ABB RobotStudio station: Material Handeling (First Class) (5-3-2024)@7020.rsstn

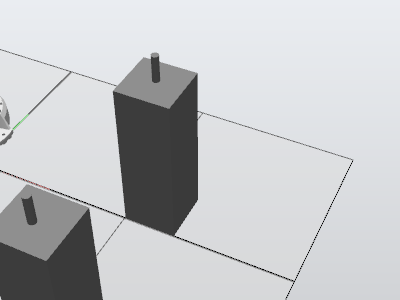
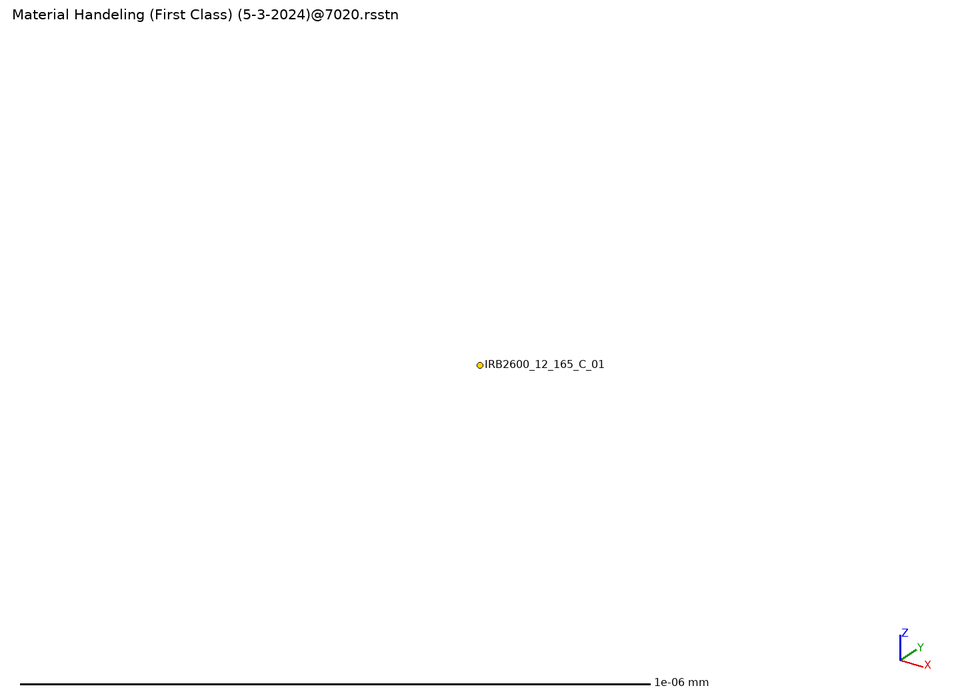
[picture v1: parts stored in the station drawn from their meshes, with robot base, taught points and paths (robot models come from the ABB library and are not in the file)]
Station Station (saved by RobotStudio 22.3.10141.1)
Controller Controller24, task T_ROB1: task frame (RAPID world) sits at (0, 0, 290) mm in the station
Controller Controller24
  mechanical unit ROB_1: IRB2600_12_165_C_01, 6 joints, base frame (0, 0, 0) mm
Layout (positions relative to the parent item):
  - Robot Base [part, from Robotics 7020\Cement Base.rslib] at (-450, -450, 0) mm
  - IRB2600_12_165_C_01 [mechanism, from %ABB.RobotStudio.Models.IRB2600%\IRB2600_12_165_C_01.rslib] at (0, 0, 290) mm; joint values [-1.2189, 0, 0, 0, 0.5236, 0] (rad or m)
  - SmartComponent_1 [smart component]
    - Smart_Gripper_Servo_Fingers [mechanism, from Tools\ABB_Smart_Gripper_Servo_Fingers.rslib] at (351.05, -956.21, 1507.5) mm, rotated rx 180 ry 60 rz 110.16 deg; joint values [0] (rad or m)
    - Detacher [smart component, from Components\Detacher.rslib]
        properties: Child=(none); KeepPosition=true
    - Attacher [smart component, from Components\Attacher.rslib]
        properties: Parent=(none); Flange=0; Child=(none); Mount=false; Offset=[0 0 0]; Orientation=[0 0 0]
    - LogicGate [smart component, from Components\LogicGate.rslib]
        properties: Operator=NOT; Delay=0
    - JointMover [smart component, from Components\JointMover.rslib]
        properties: Mechanism=(none); Relative=false; Duration=0
    - JointMover_2 [smart component, from Components\JointMover.rslib]
        properties: Mechanism=(none); Relative=false; Duration=0
  - Piller_1 [part] at (1003.05, -982.86, 0) mm, size 300 x 300 x 900 mm
  - Piller_2 [part] at (1006.06, 0, 0) mm, size 300 x 300 x 900 mm
  - Part_8 [part] at (1141.81, -843.1, 0) mm, size 40 x 39.4 x 150 mm
  - Part_9 [part] at (1152.35, 160.25, 0) mm, size 40 x 39.4 x 150 mm
Attachment: Smart_Gripper_Servo_Fingers is attached to IRB2600_12_165_C_01 / Link6
Targets, tools, work objects and paths stored in the station, written as RAPID:
! task T_ROB1
MODULE CalibData
  PERS tooldata Servo:=[TRUE,[[0,0,114.2],[1,0,0,0]],[0.215,[8.7,12.3,49.2],[1,0,0,0],0.00021,0.00024,0.00009]];
ENDMODULE

